INTERFACE ITF_States

PROPERTY AbortingState : ITF_PackMLState
GET
END_GET
SET
END_SET
END_PROPERTY

PROPERTY MyNextState : ITF_PackMLState
GET
END_GET
SET
END_SET
END_PROPERTY

PROPERTY StoppingState : ITF_PackMLState
GET
END_GET
SET
END_SET
END_PROPERTY

END_INTERFACE

(* stored: Version 1.1.0.1, ProductVersion 3.1.4024.12
   Itf ITF_States: Id {f78a5306-5325-4b69-88ea-abfd1faa0fa6}
   Property AbortingState: Id {c8c0a174-8c19-441c-9d8f-1df88fb0d009}
   Get Get: Id {71ef9a35-c265-436a-8843-38cfee5e2c1b}
   Set Set: Id {ff67ca8f-c3bc-45d9-8dfc-3add97352aec}
   Property MyNextState: Id {77c172a3-417a-4994-8780-12aa237315d1}
   Get Get: Id {ecc05414-002f-4497-8d83-1198c48115fa}
   Set Set: Id {6ff3c9f2-ff7c-4166-8211-e2fbc88eae3f}
   Property StoppingState: Id {22e9742a-6075-4c8b-89a5-61d3e905a7ea}
   Get Get: Id {49c4a6f8-9363-4697-a498-1c53f172da7e}
   Set Set: Id {fbe9b580-0db2-4479-8559-e45ee5231514} *)
